FUNCTION_BLOCK RandomGenerator (* Basic Function Block Type *)
  (* Standard: 61499-2 *)
  (* Version 0.0, 8/30/2016, Dmitry, nxtControl GmbH, Template *)
  PACKAGE Main;
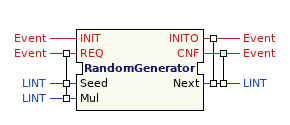
  EVENT_INPUT
    INIT; (* Initialization Request *)
    REQ WITH Seed, Mul; (* Normal Execution Request *)
  END_EVENT
  EVENT_OUTPUT
    INITO WITH Next; (* Initialization Confirm *)
    CNF WITH Next; (* Execution Confirmation *)
  END_EVENT
  VAR_INPUT
    Seed : LINT;
    Mul : LINT;
  END_VAR
  VAR_OUTPUT
    Next : LINT; (* Next random number *)
  END_VAR
  VAR
    Cur : LINT;
    OldSeed : LINT;
  END_VAR
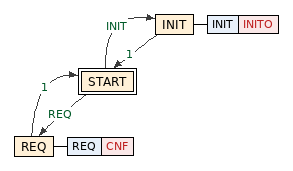
  EC_STATES
    START; (* Initial State *)
    INIT : INIT -> INITO; (* Initialization *)
    REQ : REQ -> CNF; (* Normal execution *)
  END_STATES
  EC_TRANSITIONS
    START TO INIT := INIT;
    INIT TO START := 1;
    START TO REQ := REQ;
    REQ TO START := 1;
  END_TRANSITIONS
  ALGORITHM INIT IN ST: (* Initialization algorithm *)
OldSeed := Seed;
Cur := OldSeed;
  END_ALGORITHM
  ALGORITHM REQ IN ST: (* Normally executed algorithm *)
IF OldSeed <> Seed THEN
	OldSeed := Seed;
	Cur := OldSeed;
END_IF;

Cur := (Cur * Mul + 3217587316749923) * 4 / 1024;
Next := Cur;
  END_ALGORITHM
END_FUNCTION_BLOCK
